# B&R Automation Studio project boxLift
Automation Studio 4.12.6.106; technology packages: mapp 5.24.2, mappView 5.24.2

## Configuration Config1

CPU X20CP1586, AutomationRuntime B4.93, Build 4.1.2, Vc V4.72.6

CPU X20CP1686X, AutomationRuntime J4.93, Build 4.1.2, Vc V4.73.2

### Task classes (Cpu.sw)
```
Cyclic#4:
  SimConnect <- SimConnect.prg
  Program <- Program.prg
Libraries: standard
```

### Hardware
```
X20CP1686X : X20CP1686X v1.8.2.0
  Connector IF2:
    ActivateDevice = 1
  ConfigurationID = boxLift_Config1
  Simulation = 1
  FileDevice1
  FileDeviceName1 = Location
  FileDevicePath1 = C:\TEMP\
  ActivateOpcUa = 1
  OpcUaInformationModels_PV_Version = 1
```

### PvMap.vvm - X20CP1686X/PvMap.vvm
```iecst
VAR_CONFIG
	Cyclic#1.::SimConnect:Inputs.diLiftPosTop AT %Q.Cyclic#1.::Program:Lift.Status.diLiftTop; (*Insert your comment here...*)
	Cyclic#1.::SimConnect:Inputs.diLiftPosUnload AT %Q.Cyclic#1.::Program:Lift.Status.diLiftUnload; (*Insert your comment here...*)
	Cyclic#1.::SimConnect:Inputs.diLiftPosBottom AT %Q.Cyclic#1.::Program:Lift.Status.diLiftBot; (*Insert your comment here...*)
	Cyclic#1.::SimConnect:Inputs.diBoxLift AT %Q.Cyclic#1.::Program:Lift.Status.diBoxLift; (*Insert your comment here...*)
	Cyclic#1.::SimConnect:Inputs.diBoxBottom AT %Q.Cyclic#1.::Program:Conv.Status.diConvBot; (*Insert your comment here...*)
	Cyclic#1.::SimConnect:Inputs.diBoxUnload AT %Q.Cyclic#1.::Program:Conv.Status.diBoxUnload; (*Insert your comment here...*)
	Cyclic#1.::SimConnect:Inputs.diBoxTop AT %Q.Cyclic#1.::Program:Conv.Status.diConvTop; (*Insert your comment here...*)
	Cyclic#1.::Program:Lift.Cmd.doLiftTop AT %Q.Cyclic#1.::SimConnect:Outputs.doLiftTop; (*Insert your comment here...*)
	Cyclic#1.::Program:Lift.Cmd.doLiftUnload AT %Q.Cyclic#1.::SimConnect:Outputs.doLiftUnload; (*Insert your comment here...*)
	Cyclic#1.::Program:Conv.Cmd.doConvTop AT %Q.Cyclic#1.::SimConnect:Outputs.doConvTop; (*Insert your comment here...*)
	Cyclic#1.::Program:Lift.Cmd.doLiftBot AT %Q.Cyclic#1.::SimConnect:Outputs.doLiftBottom; (*Insert your comment here...*)
	Cyclic#1.::Program:Lift.Cmd.doConvLift AT %Q.Cyclic#1.::SimConnect:Outputs.doConvLift; (*Insert your comment here...*)
	Cyclic#1.::Program:Conv.Cmd.doConvBot AT %Q.Cyclic#1.::SimConnect:Outputs.doConvBottom; (*Insert your comment here...*)
	Cyclic#1.::SimConnect:Inputs.diLiftPosTop AT %Q.Cyclic#1.::AlarmHandl:diLiftTop; (*Insert your comment here...*)
	Cyclic#1.::SimConnect:Inputs.diLiftPosBottom AT %Q.Cyclic#1.::AlarmHandl:diLiftBot; (*Insert your comment here...*)
	Cyclic#1.::SimConnect:Inputs.diBoxTop AT %Q.Cyclic#1.::AlarmHandl:diBoxTop; (*Insert your comment here...*)
	Cyclic#1.::SimConnect:Inputs.diBoxBottom AT %Q.Cyclic#1.::AlarmHandl:diBoxBot; (*Insert your comment here...*)
	Cyclic#1.::SimConnect:Inputs.diBoxUnload AT %Q.Cyclic#1.::AlarmHandl:diBoxUnload; (*Insert your comment here...*)
END_VAR
```

### BoxAla.mpalarmxcore - X20CP1686X/mappServices/BoxAla.mpalarmxcore
```
Element MpLinkBOXgAlarmXCore (Type=mpalarmxcore)
  mapp.AlarmX.Core.Configuration:
    [0]:
      Name = BoxLost
      Message = A box was not deliivered
      Code = 117
      Behavior = PersistentAlarm
```

### BoxAlaHis.mpalarmxhistory - X20CP1686X/mappServices/BoxAlaHis.mpalarmxhistory
```
Element MpLinkBOXgAlarmXHistory (Type=mpalarmxhistory)
```

### Config.mpalarmxcore - X20CP1686X/mappServices/Config.mpalarmxcore
```
Element gAlarmXCore (Type=mpalarmxcore)
  mapp.AlarmX.Core.Configuration:
    [0]:
      Name = BoxLost
      Message = A box is lost
      Code = 117
      Severity = 10
      Behavior = PersistentAlarm
```

### Core.mpalarmxcore - X20CP1686X/mappServices/Core.mpalarmxcore
```
Element gAlarmXCore (Type=mpalarmxcore)
  mapp.AlarmX.Core:
    Mapping:
      [0]:
        Alarm = BoxLost
        [0] = Reaction
          Name = StopAll
  mapp.AlarmX.Core.Configuration:
    [0]:
      Name = BoxLost
      Message = A box is lost
      Code = 117
      Severity = 10
      Behavior = PersistentAlarm
    [1]:
      Name = TestingAlarm
      Message = Testing Alarm
      Behavior = PersistentAlarm
```

## Logical view

Binary libraries used (declarations not repeated): operator, runtime, astime, AsIecCon, standard, MpCom, MpAlarmX, MpBase, MpServer

### Global.typ - Global data types
```iecst
TYPE
    StatesEnum:
	(
		WAIT,
		TOP_POSE,
		BOT_POSE,
		GET_BOX,
		UNLOAD_POSE,
		UNLOAD_BOX
	);

    MainType : STRUCT
        AutomaticControl : BOOL := TRUE;
        State : StatesEnum := WAIT;
		Error : BOOL;
        Restart : BOOL;
    END_STRUCT;

END_TYPE
```

### Global.var - Global variables
```iecst
VAR
    gMain : MainType;
END_VAR

VAR CONSTANT

END_VAR
```


### Program Logical/SimConnect (IEC)

#### Types.typ
```iecst
TYPE
	SimParamsType : 	STRUCT  (*Parameters for RobotStudio simulation and internal .*)
		aoBoxSpawnRateTop : REAL; (*Spawn rate for boxes at top conveyor.*)
		aoBoxSpawnRateBottom : REAL; (*Spawn rate for boxes at bottom conveyor.*)
		aoConvSpeedInTop : REAL; (*Speed for ingoing conveyor top.*)
		aoConvSpeedOutTop : REAL; (*Speed for outgoing top conveyor.*)
		aoConvSpeedInBottom : REAL; (*Speed for ingoing bottom conveyor.*)
		aoConvSpeedOutBottom : REAL; (*Speed for outgoing bottom conveyor.*)
		aoConvSpeedLift : REAL; (*Speed for lift conveyor.*)
		aoConvSpeedUnload : REAL; (*Speed for unoad conveyor.*)
		aoLiftTravelSpeed : REAL; (*Travel speed between positions for the lift.*)
		diLastExtCounter : UDINT; (*Last value of the external counter.*)
		InternalHeartbeatTimer : TOF; (*Used for internal heartbeat.*)
		HeartbeatTimer : TOF; (*Used for heartbeat monitoring.*)
	END_STRUCT;
	ASInputsType : 	STRUCT  (*Inputs from OPC UA node to Automation Studio.*)
		diBoxTop : BOOL := FALSE; (*Box at top conveyor unload position.*)
		diBoxBottom : BOOL := FALSE; (*Box at bottom conveyor unload position.*)
		diBoxLift : BOOL := FALSE; (*Box loaded on lift.*)
		diBoxUnload : BOOL := FALSE; (*Box at unload conveyor.*)
		diLiftPosTop : BOOL := FALSE; (*Lift at top position.*)
		diLiftPosBottom : BOOL := FALSE; (*Lift at bottom position.*)
		diLiftPosUnload : BOOL := FALSE; (*Lift at unload position.*)
		diSimRunning : BOOL := FALSE; (*Indicates active simulation.*)
		aiExternalCounter : UDINT := 0; (*External heartbeat counter.*)
	END_STRUCT;
	ASOutputsType : 	STRUCT  (*Outputs from SimConnect task to OPC UA node (and/or other tasks).*)
		doLiftTop : BOOL := FALSE; (*Move lift to top position.*)
		doLiftBottom : BOOL := FALSE; (*Move lift to bottom position.*)
		doLiftUnload : BOOL := FALSE; (*Move lift to unload position.*)
		doConvTop : BOOL := FALSE; (*Top conveyor on/off.*)
		doConvBottom : BOOL := FALSE; (*Bottom conveyor on/off.*)
		doConvLift : BOOL := FALSE; (*Lift conveyor on/off.*)
		doInternalHeartbeat : BOOL := FALSE; (*Internal heartbeat.*)
		doConnectionError : BOOL := FALSE; (*Indicates an error with OPC UA connection.*)
	END_STRUCT;
END_TYPE
```

#### Variables.var
```iecst
VAR
	Inputs : ASInputsType; (*Inputs from OPC UA node to Automation Studio.*)
	Outputs : ASOutputsType; (*Outputs from Automation Studio to OPC UA node.*)
	Configuration : SimParamsType; (*Simulation parameters for Robot Studio.*)
END_VAR
```

#### Main.st
```iecst
PROGRAM _INIT
	(* 	These parameters can be changed to change
	 	the behaviour of the simulation.
	 	Default values and units are commented after each parameter. *)
	Configuration.aoBoxSpawnRateTop			:= 20; (* 20 s *)
	Configuration.aoBoxSpawnRateBottom		:= 25; (* 25 s *)
	Configuration.aoConvSpeedInTop			:= 0.6; (* 0.6 m/s *)
	Configuration.aoConvSpeedOutTop			:= 0.7; (* 0.9 m/s *)
	Configuration.aoConvSpeedInBottom		:= 0.5; (* 0.5 m/s *)
	Configuration.aoConvSpeedOutBottom		:= 0.7; (* 0.9 m/s *)
	Configuration.aoConvSpeedLift			:= 0.9; (* 0.9 m/s *)
	Configuration.aoConvSpeedUnload			:= 0.9; (* 0.9 m/s *)
	Configuration.aoLiftTravelSpeed			:= 0.6; (* 0.4 m/s *)

	(* 	The global variables to communicate with OPC UA has to be initated.
	Don't change anything below! *)
	Inputs;
	Outputs;

	(* Initiate counter and heartbeat timer. *)
	Configuration.InternalHeartbeatTimer(IN:=TRUE, PT:=T#500ms);
	Configuration.HeartbeatTimer(IN:=TRUE, PT:=T#1500ms);

END_PROGRAM

PROGRAM _CYCLIC
	(*	The heartbeat is used to check if the OPC UA connection between
		Automation Studio and RobotStudio is still up.
		In both AS and RS, a counter is increased once per second,
		and if the difference between the internal and incoming
		counter is greater than the tolerance, it is assumed that the
		OPC UA connection is down. *)

	(*	Call and update internal counter only when the simulation is active. *)
	IF Inputs.diSimRunning THEN

		IF NOT Configuration.HeartbeatTimer.Q THEN

			(* 	If the current external counter is the same as the last one,
				the connection is down. *)
			IF Inputs.aiExternalCounter = Configuration.diLastExtCounter THEN
				Outputs.doConnectionError := TRUE;
			ELSE
				Configuration.diLastExtCounter := Inputs.aiExternalCounter;
				Outputs.doConnectionError := FALSE;
			END_IF

		END_IF

	END_IF

	(* Update counter and call timer. *)
	Outputs.doInternalHeartbeat := Configuration.InternalHeartbeatTimer.Q;
	Configuration.InternalHeartbeatTimer(IN:=(NOT Configuration.InternalHeartbeatTimer.Q), PT:=T#500ms);
	Configuration.HeartbeatTimer(IN:=(NOT Configuration.HeartbeatTimer.Q), PT:=T#1500ms);

END_PROGRAM

PROGRAM _EXIT

END_PROGRAM
```

- Visualisation Logical/mappView (not shown)

### Program Logical/Program (IEC)

#### Types.typ
```iecst
TYPE
	ConvType : STRUCT
		Cmd : ConvControlType;
		Status : ConvStatusType;
	END_STRUCT;

	ConvControlType : STRUCT
		doConvTop : BOOL := TRUE;
		doConvBot : BOOL := TRUE;
	END_STRUCT;

	ConvStatusType : STRUCT
		diConvBot : BOOL := FALSE;
		diConvTop : BOOL := FALSE;
		diBoxUnload : BOOL := FALSE;
	END_STRUCT;

	LiftType : STRUCT
		Cmd : LiftControlType;
		Status : LiftStatusType;
	END_STRUCT;

	LiftControlType : STRUCT
		doLiftTop : BOOL := FALSE;
		doLiftBot : BOOL := FALSE;
		doConvLift : BOOL := FALSE;
		doLiftUnload : BOOL := FALSE;
	END_STRUCT;

	LiftStatusType : STRUCT
		diLiftBot : BOOL := FALSE;
		diLiftTop : BOOL := FALSE;
		diBoxLift : BOOL := FALSE;
		diLiftUnload : BOOL := FALSE;
	END_STRUCT;

END_TYPE
```

#### Variables.var
```iecst
VAR
	Conv : ConvType;
	Lift : LiftType;

	NextPose : StatesEnum;
	selectLift : StatesEnum;

	Input : BOOL;
	Output : BOOL;
END_VAR
```

#### Cyclic.st
```iecst
(*
Pseudo Code
	cases = [ConvTop, ConvBot]

	Case 1:
	if diConvTop == True:
		doConvTop = False;
		doLiftTop = True;
		Unload;
	Case 2:
	if diConvBot == True:
		doConvBot = False;
		doLiftBot = True;

			while diLiftUnload == False;
				doLiftUnload = True;

	if currently doing somehting
		place in queue

	*)

// VAR
// 	TYPE
		// Conv : STRUCT
		// 	CmdType : ConvOutputs
		// 	Status : ConvInputs;
		// END_STRUCT

		// ConvOutputs : STRUCT
		// 	doConvTop : BOOL := FALSE;
		// 	doConvBot : BOOL := FALSE;
		// END_STRUCT

		// ConvInputs : STRUCT
		// 	diConvBot : BOOL := FALSE;
		// 	diConvTop : BOOL := FALSE;
		// 	diBoxtUnload : BOOL := FALSE;
		// END_STRUCT

		// Lift : STRUCT
		// 	Cmd : LiftOutputs;
		// 	Status : LiftrInputs;
		// END_STRUCT

		// LiftOutputs : STRUCT
		// 	doLiftTop : BOOL := FALSE;
		// 	doLiftBot : BOOL := FALSE;
		// 	doConvLift : BOOL := FALSE;
		// 	doLiftUnload : BOOL := FALSE;
		// END_STRUCT

		// LiftInputs : STRUCT
		// 	diLiftBot : BOOL := FALSE;
		// 	diLiftTop : BOOL := FALSE;
		// 	diBoxLift : BOOL := FALSE;
		// 	diLiftUnload : BOOL := FALSE;
		// END_STRUCT

		// StatesEnum:
		// (
		// 	TOP_POSE,
		// 	BOT_POSE,
		// 	GET_BOX,
		// 	UNLOAD_POSE,
		// 	UNLOAD_BOX,
		// 	WAIT
		// );
// 	END_TYPE
// END_VAR

PROGRAM _CYCLIC

	IF MpAlarmXCheckReaction(gAlarmXCore, 'StopAll') THEN
		Input := TRUE;
	ELSE
		Input := FALSE;
	END_IF;

	IF EDGEPOS(Input) THEN
		Conv.Cmd.doConvBot := FALSE;
		Conv.Cmd.doConvTop := FALSE;
		Lift.Cmd.doLiftBot := FALSE;
		Lift.Cmd.doLiftTop := FALSE;
		Lift.Cmd.doLiftUnload := FALSE;
		Lift.Cmd.doConvLift := FALSE;
		selectLift := gMain.State;

	ELSIF EDGENEG(Input) THEN
		Conv.Cmd.doConvTop := TRUE;
		Conv.Cmd.doConvBot := TRUE;
	END_IF;

	IF NOT MpAlarmXCheckReaction(gAlarmXCore, 'StopAll') THEN
		IF gMain.AutomaticControl THEN

			IF (Conv.Status.diConvTop AND NOT Lift.Status.diLiftTop) THEN
				NextPose := TOP_POSE;
				Conv.Cmd.doConvTop := FALSE;
			END_IF;

			IF (Conv.Status.diConvBot = TRUE AND NOT Lift.Status.diLiftBot) THEN
				NextPose := BOT_POSE;
				Conv.Cmd.doConvBot := FALSE;
			END_IF;

			IF EDGEPOS(gMain.Restart) THEN
				selectLift := WAIT;
				gMain.Restart := FALSE;
			END_IF;

			gMain.State := selectLift;

			CASE selectLift OF

				WAIT:
					IF Conv.Status.diConvTop = TRUE THEN
							selectLift := TOP_POSE;
						Conv.Cmd.doConvTop := FALSE;
					ELSIF (Conv.Status.diConvBot = TRUE) THEN
						selectLift := BOT_POSE;
						Conv.Cmd.doConvBot := FALSE;
					END_IF;

				TOP_POSE:
					Lift.Cmd.doLiftTop := TRUE;
					IF Lift.Status.diLiftTop THEN
						Lift.Cmd.doLiftTop := FALSE;
						Conv.Cmd.doConvTop := TRUE;
						selectLift := GET_BOX;
					END_IF;

				BOT_POSE:
					Lift.Cmd.doLiftBot := TRUE;
					IF Lift.Status.diLiftBot THEN
						Lift.Cmd.doLiftBot := FALSE;
						Conv.Cmd.doConvBot := TRUE;
						selectLift := GET_BOX;
					END_IF;

				GET_BOX:
					Lift.Cmd.doConvLift := TRUE;
					IF Lift.Status.diBoxLift = TRUE THEN //the box is succesfully loaded onto the lift
						Lift.Cmd.doConvLift := FALSE;
						selectLift := UNLOAD_POSE;
					END_IF;

				UNLOAD_POSE:
					Lift.Cmd.doLiftUnload := TRUE;
					IF Lift.Status.diLiftUnload THEN
						Lift.Cmd.doLiftUnload := FALSE;
						selectLift := UNLOAD_BOX;
					END_IF;

				UNLOAD_BOX:
					Lift.Cmd.doConvLift := TRUE;
					IF Conv.Status.diBoxUnload THEN
						Lift.Cmd.doConvLift := FALSE;
						selectLift := WAIT;
					END_IF;
			END_CASE;
		END_IF;
	END_IF;
END_PROGRAM
```

#### Init.st
```iecst
PROGRAM _INIT
	(* Insert code here *)
	Conv.Cmd.doConvBot := TRUE;
	Conv.Cmd.doConvTop := TRUE;
END_PROGRAM
```

### Program Logical/AlarmHandler (IEC)

#### Types.typ
```iecst
TYPE
	SystemManagementType : STRUCT
		InputSignals : InputSignals;
		CurrentActions : CurrentActionsType;
	END_STRUCT;

	CurrentActionsType : STRUCT
		GettingTop : BOOL;
		GettingBot : BOOL;
	END_STRUCT;

	InputSignalsType : STRUCT
		diBoxTop : BOOL;
		diBoxBot : BOOL;
		diLiftTop : BOOL;
		diLiftBot : BOOL;
		diBoxUnload : BOOL;
	END_STRUCT;

	ErrorManagementType : STRUCT
		BoxCounter : BoxCounterType;
		TimerCounter : TimerCounterType;
		Conditions : ConditionsType;
		ErrorCommands : ErrorCommandsType;
	END_STRUCT;

	ConditionsType : STRUCT
		ConditionTopErr : BOOL;
		ConditionBotErr : BOOL;
	END_STRUCT;

	TimerCounterType : STRUCT
		TON_0 : TON;
		TON_1 : TON;
	END_STRUCT;

	BoxCounterType : STRUCT
		BoxDeliveredCnt : CTU;
		BoxArrivedCnt : CTU;
		BoxesReceived : UINT;
	END_STRUCT;

	ErrorCommandsType : STRUCT
		CauseError : BOOL;
		CauseTestError : BOOL;
		ResetAlarms : BOOL;
		ClearHistory : BOOL;
		AcknowledgeAlarms : BOOL;
	END_STRUCT;

END_TYPE
```

#### Variables.var
```iecst
VAR
	diBoxTop : BOOL;
	diBoxBot : BOOL;
	diLiftTop : BOOL;
	diLiftBot : BOOL;
	diBoxUnload : BOOL;
	NewBox : BOOL;
	BoxDeliveredCnt : CTU;
	BoxArrivedCnt : CTU;
	GettingTop : BOOL;
	GettingBot : BOOL;
	ConditionTopErr : BOOL;
	ConditionBotErr : BOOL;
	TON_0 : TON;
	TON_1 : TON;
	BoxesReceived : UINT;
	MpAlarmXCore_0 : MpAlarmXCore;
	MpAlarmXHistory_0 : MpAlarmXHistory;
    MpAlarmXAcknowledgeAll_0 : MpAlarmXAcknowledgeAll;
	AlarmLanguage : STRING[20] := 'en|metric';

    CauseError : BOOL;
    CauseTestError : BOOL;
    ResetAlarms : BOOL;
    ClearHistory : BOOL;
    AcknowledgeAlarms : BOOL;
END_VAR

VAR CONSTANT

END_VAR
```

#### Cyclic.st
```iecst
(*
Psuedo code:

// check how many boxes have arrived?

if diTopBox:
	BoxArrived++:
if diBotBox:
	BoxArrived++;
if diUnload:
	BoxDeleivered++;

if lift called:
	start timer;
if enough time passed && diUnload not true:
	box failed TO be delivered;
	raise alarm;
ELSE IF diUnload is TRUE:
	reset timer;

8s for top
5s for bot

 *)

PROGRAM _CYCLIC

	MpAlarmXCore_0();
	MpAlarmXHistory_0();
	MpAlarmXAcknowledgeAll_0();
	MpAlarmXHistory_0.Language := ADR(AlarmLanguage);

	NewBox := diBoxBot OR diBoxTop;
	BoxArrivedCnt(CU:=NewBox);

	IF gMain.State = TOP_POSE THEN
		GettingTop := TRUE;
	ELSIF gMain.State = BOT_POSE THEN
		GettingBot := TRUE;
	END_IF;

	TON_0(IN:=GettingTop, PT:=T#13s);
	TON_1(IN:=GettingBot, PT:=T#13s);

	IF diBoxUnload THEN
		GettingTop := FALSE;
		GettingBot := FALSE;
	END_IF;

	BoxDeliveredCnt(CU:=diBoxUnload);

	ConditionTopErr := GettingTop AND TON_0.Q;
	ConditionBotErr := GettingBot AND TON_1.Q;

	IF ConditionBotErr OR ConditionTopErr OR CauseError THEN
		IF NOT MpAlarmXCheckReaction(gAlarmXCore, 'StopAll') THEN
			MpAlarmXSet(gAlarmXCore, 'BoxLost');
		END_IF;
		gMain.Error := TRUE;
		gMain.State := WAIT;
	END_IF;

	IF AcknowledgeAlarms THEN
		MpAlarmXAcknowledge(gAlarmXCore, 'BoxLost');
		MpAlarmXAcknowledge(gAlarmXCore, 'TestingAlarm');
	END_IF;

	IF CauseTestError THEN
		MpAlarmXSet(gAlarmXCore, 'TestingAlarm');
	END_IF;

	IF ResetAlarms THEN
		MpAlarmXReset(gAlarmXCore, 'BoxLost');
		MpAlarmXReset(gAlarmXCore, 'TestingAlarm');
		GettingTop := FALSE;
		GettingBot := FALSE;
		gMain.Restart := TRUE;
	END_IF;

	IF ClearHistory THEN
		MpAlarmXClearHistory(gAlarmXHistory);
	END_IF;

	BoxesReceived := BoxDeliveredCnt.CV;

END_PROGRAM
```

#### Exit.st
```iecst
PROGRAM _EXIT
	MpAlarmXCore_0.Enable := FALSE;
	MpAlarmXCore_0();

	 MpAlarmXHistory_0.Enable := FALSE;
	 MpAlarmXHistory_0();

END_PROGRAM
```

#### Init.st
```iecst
PROGRAM _INIT
	MpAlarmXCore_0.Enable := TRUE;
	MpAlarmXCore_0.MpLink := ADR(gAlarmXCore);

	MpAlarmXAcknowledgeAll_0.Enable := TRUE;
	MpAlarmXAcknowledgeAll_0.MpLink := ADR(gAlarmXCore);

	MpAlarmXHistory_0.Enable := TRUE;
	MpAlarmXHistory_0.MpLink := ADR(gAlarmXHistory);
	MpAlarmXHistory_0.DeviceName := ADR('Location');

END_PROGRAM
```

#### Main.st
```iecst
PROGRAM _INIT
	MpAlarmXCore_0.Enable := TRUE;
	MpAlarmXCore_0.MpLink := ADR(MpLinkBOXgAlarmXCore);

END_PROGRAM

(*
Psuedo code:

// check how many boxes have arrived?

IF diTopBox:
	BoxArrived++:
IF diBotBox:
	BoxArrived++;
IF diUnload:
	BoxDeleivered++;

IF lift called:
	start timer;
IF enough time passed && diUnload NOT TRUE:
	box failed TO be delivered;
	raise alarm;
else if diUnload is true:
	reset timer;

8s for top
5s for bot

 *)

PROGRAM _CYCLIC

	MpAlarmXCore_0();
	//MpAlarmXHistory_0.Language := AlarmLanguage;

	NewBox := diBoxBot OR diBoxTop;
	BoxArrivedCnt(CU:=NewBox);

	IF diBoxTop THEN
		GettingTop := TRUE;
	ELSIF diBoxBot THEN
		GettingBot := TRUE;
	END_IF;

	TON_0(IN:=GettingTop, PT:=T#13s);
	TON_1(IN:=GettingBot, PT:=T#13s);

	IF diBoxUnload THEN
		GettingTop := FALSE;
		GettingBot := FALSE;
	END_IF;

	BoxDeliveredCnt(CU:=diBoxUnload);

	ConditionTopErr := GettingTop AND TON_0.Q;
	ConditionBotErr := GettingBot AND TON_1.Q;

	IF ConditionBotErr OR ConditionTopErr THEN
		// MpAlarmXSet(MpLinkBOXgAlarmXCore, 'BoxLost');
		gError := TRUE;
	END_IF;

	BoxesReceived := BoxDeliveredCnt.CV;

END_PROGRAM

PROGRAM _EXIT
	MpAlarmXCore_0.Enable := FALSE;
	MpAlarmXCore_0();

END_PROGRAM
```

### Program Logical/Testing

#### Variables.var
```iecst
VAR
	Input : BOOL;
	Output : BOOL;
	R_TRIG_0 : R_TRIG;
	F_TRIG_0 : F_TRIG;
END_VAR
```

#### Main.st
```iecst
PROGRAM _INIT
	Output := TRUE;

END_PROGRAM

PROGRAM _CYCLIC
	R_TRIG_0(CLK := Input);
	F_TRIG_0(CLK := Input);

	IF R_TRIG_0.Q THEN
		Output := FALSE;
	ELSIF F_TRIG_0.Q THEN
		Output := TRUE;
	END_IF;

END_PROGRAM

PROGRAM _EXIT
	(* Insert code here *)
END_PROGRAM
```
